// TIA Portal V17 export
// export: Created 2025-03-07T09:18:36.4180045Z, ExportSetting WithDefaults, DisplayName Totally Integrated Automation Portal, DisplayVersion V17 Update 8, DisplayName TIA Portal Openness, DisplayVersion V17 Update 8, DisplayName TIA Portal Version Control Interface, DisplayVersion V17, DisplayName SINAMICS Startdrive Advanced, DisplayVersion V17 SP2, DisplayName SINAMICS Startdrive G110M, G120, G120C, G120D, G120P, G115D, DisplayVersion V17 SP2, DisplayName SINAMICS Startdrive G130, G150, S120, S150, SINAMICS MV, S210, DisplayVersion V17 SP2, DisplayName STEP 7 Professional, DisplayVersion V17 Update 8, DisplayName SINUMERIK ONE STEP 7 Toolbox, DisplayVersion V17 Update 12, DisplayName SINUMERIK 840D sl STEP 7 Toolbox, DisplayVersion V17 Update 12, DisplayName STEP 7 Safety, DisplayVersion V17 Update 6, DisplayName WinCC Advanced, DisplayVersion V17 Update 8
DATA_BLOCK "DB1017_SAFETY_DOORS_LOAD_UNLOAD"   // DB1017, F_DB
{ DB_Accessible_From_OPC_UA := 'FALSE' }
AUTHOR : ETXETAR
VERSION : 1.0
// stored: AutoNumber false, DBAccessibleFromOPCUA false, DBAccessibleFromWebserver true, InstanceOfName FB1016_SAFETY_DOORS, InstanceOfType FB
"FB1016_SAFETY_DOORS"
   // VAR_INPUT
   //    FEEDBACK_OFF_SAFETY_DOORS_IN : Bool;
   //    FEEDBACK_OFF_E_SAFE_DOORS_RST_STR_IN : Bool;
   //    DOOR_1 : Bool;
   //    DOOR_2 : Bool;
   //    DOOR_3 : Bool;
   //    DOOR_4 : Bool;
   //    DOOR_5 : Bool;
   //    DOOR_6 : Bool;
   //    DOOR_7 : Bool;
   //    DOOR_8 : Bool;
   //    DOOR_9 : Bool;
   //    DOOR_10 : Bool;
   // END_VAR
   // VAR_OUTPUT
   //    SAFE_DOORS_CLOSED_LOCKED : Bool;
   //    SAFE_DOORS_CLOSED_LOCKED_DEL2 : Bool;
   //    SAFE_DOORS_CLOSED_LOCKED_DEL3 : Bool;
   //    SAFE_DOORS_CLOSED_LOCKED_DEL4 : Bool;
   //    FEEDBACK_ERROR : Bool;
   // END_VAR
   // VAR
   //    ALL_DOORS_CLOSED_AND_LOCKED : Bool;
   //    SAFE_GATES_CLOSED_AND_LOCKED_RESET : Bool;
   //    SAFE_GATES_CLOSED_AND_LOCKED_RESET_REQ : Bool;
   //    FEEDBACK_OFF_OK : Bool;
   //    SFDOOR_Instance : SFDOOR;
   //    F_DOOR_DEL2_Timer_Instance : TOF;
   //    F_DOOR_DEL3_Timer_Instance : TOF;
   //    F_DOOR_DEL4_Timer_Instance : TOF;
   //    FDBACK_Instance : FDBACK;
   //    F_IEC_Timer_FEEDBACK : TON;
   // END_VAR
BEGIN
END_DATA_BLOCK
